(* IEC 61131-3 sources: codesys-build/examples/frame-assembly/src/transport/FB_Conveyor/methods, 1 file *)

(* ---- SetEnabled.st ---- *)
METHOD PUBLIC SetEnabled
VAR_INPUT
	Asserted : BOOL;
END_VAR
VAR_INST
	Calls : UDINT;
END_VAR
Enabled := Asserted;
Calls := Calls + 1;
END_METHOD
